(* Logix 5000 project; controller cal1632 1756-L62 rev 16.20; software revision 16.05; part 53 of 61 *)
(* tags used below, declared in another part *)
   turret_wa_pos_doff_request : BOOL;   // Turret Move to Winder A Doff Position Request
   turret_wa_pos_run_request : BOOL;   // Turret Move to Winder A Run Position
   turret_wb_pos_doff_request : BOOL;   // Turret Move to Winder B Doff Position Request
   turret_wb_pos_run_request : BOOL;   // Turret Move to Winder B Run Position
   any_jog_wa_permissive : BOOL;   // Winder A Any Jog Permissive
   any_jog_wb_permissive : BOOL;   // Winder B Any Jog Permissive
   di_mode_doff : BOOL;   // Doff Mode
   di_mode_run : BOOL;   // Run Mode
   FAULT : BOOL;
   HMI : BOOL;
   p00_wac_position_pct : REAL;   // Winder Accumulator Carriage Position Filtered [% of Stroke]
   p01_recipe_active : recipe;
   p01r09_pb_global_reset : BOOL;
   p01r13_line_running : BOOL;
   p01r13_line_slow_ramp : BOOL;
   p01r13_winder_tension_ok : BOOL;
   p02_real_from_hmi : hmi_real;
   p21r10_index_kd : REAL;
   p21r10_index_ki : REAL;
   p21r10_index_kp : REAL;
   p25_ao_selected_speed : REAL;
   p29_ai_wa_speed : REAL;
   p29_ai_wa_torque : REAL;
   p29_ai_wdr_lc : REAL;
   p29_di_wdr_a : BOOL;
   p29_di_wdr_index_fwd : BOOL;
   p29_dint_to_hmi : DINT[16];
   p29_param_acc_park_sp : REAL;   // Winder Accumulator Speed Trim Park Setpoint - Where the Carriage Sits [% of Stroke]
   p29_param_acc_trim_gain : REAL;   // Winder Accumulator Speed Trim Proportional Gain Fraction of Line Speed per % of Stroke
   p29_param_index_trim_fpm : REAL;
   p29_param_speed_trim_max : REAL;
   p29_param_speed_trim_min : REAL;   // Winder Accumulator Speed Trim Minimum - Fraction of Line Speed
   p29r01 : routine;
   p29r07 : routine;
   p29r07_timer_fault : TIMER[4];
   p29r07_timer_warning : TIMER[4];
   p29r08 : routine;
   p29r08_timer_fault : TIMER[4];
   p29r08_timer_warning : TIMER[4];
   p29r09 : routine;
   p29r09_mode_doff_auto : BOOL;   // Winder Mode Doff Position - AUTO Winder A/B doff PB indexes the turret to the preset doff position
   p29r09_mode_doff_manual : BOOL;   // Winder Mode Doff Position - MANUAL Operator jogs the turret to doff, doff PBs do nothing
   p29r09_tension_mode : BOOL;
   p29r09_timer_fault : TIMER[4];
   p29r09_timer_warning : TIMER[4];
   p29r09_torque_mode : BOOL;
   p29r09_winder_a_active : BOOL;
   p29r09_winder_b_active : BOOL;
   p29r10 : routine;
   p29r10_acc_pstn_error : REAL;   // Winder Winder A Accumulator Position Error position - park setpoint [% of Stroke]
   p29r10_accel_bias : REAL;
   p29r10_calc_speed_offset : REAL;
   p29r10_index_active : BOOL;
   p29r10_line_guard : REAL;   // Winder Accumulator Speed Trim Line speed, floored at 1.0 fpm for the divide
   p29r10_misc_index_factor : REAL;
   p29r10_param_psn_gain : REAL;
   p29r10_pid_out : REAL;
   p29r10_pid_psn : PID;
   p29r10_pid_psn_cv : REAL;
   p29r10_pid_psn_pv : REAL;
   p29r10_pid_torque : REAL;
   p29r10_pid_tq : PID;
   p29r10_pid_tq_cv : REAL;
   p29r10_psn_gain : REAL;
   p29r10_request_run : BOOL;
   p29r10_run_permissive : BOOL;
   p29r10_speed_offset : REAL;
   p29r10_tension_error : REAL;   // Winder Winder A Tension Error winder_tension_sp - Load Cell [lbf]
   p29r10_timer : TIMER[4];
   p29r10_timer_fault : TIMER[4];
   p29r10_timer_warning : TIMER[4];
   p29r10_trim_clamp : sys_Limit_Clamp;   // Winder Winder A Speed Trim Clamp
   p29r10_trim_hi : REAL;   // Winder Accumulator Speed Trim Upper limit in use this scan
   p29r10_trim_lo : REAL;   // Winder Accumulator Speed Trim Lower limit in use this scan
   p29r11 : routine;
   p29r15 : routine;
   p29r15_request_jog_fwd : BOOL;
   p29r15_state : DINT;
   p29r15_wdra_active : BOOL;
   p29r16 : routine;
   p29r16_request_jog_fwd : BOOL;
   p29r17 : routine;
   p29r20 : routine;
(* P29_Winder, continued *)

ROUTINE R07_Alarms   (* ladder *)
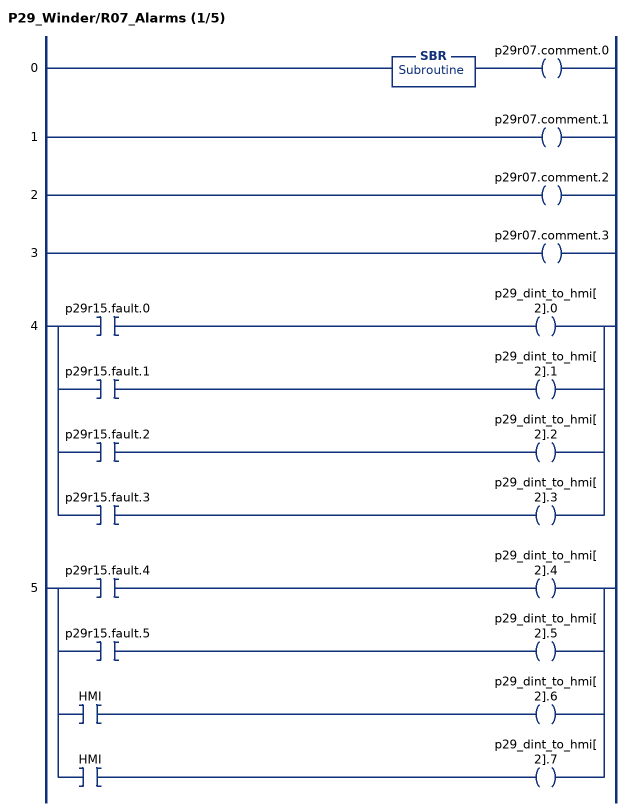
   0: SBR()OTE(p29r07.comment.0);
   1: OTE(p29r07.comment.1);
   2: OTE(p29r07.comment.2);
   3: OTE(p29r07.comment.3);
   4: [XIC(p29r15.fault.0) OTE(p29_dint_to_hmi[2].0) ,XIC(p29r15.fault.1) OTE(p29_dint_to_hmi[2].1) ,XIC(p29r15.fault.2) OTE(p29_dint_to_hmi[2].2) ,XIC(p29r15.fault.3) OTE(p29_dint_to_hmi[2].3) ];
   5: [XIC(p29r15.fault.4) OTE(p29_dint_to_hmi[2].4) ,XIC(p29r15.fault.5) OTE(p29_dint_to_hmi[2].5) ,XIC(HMI) OTE(p29_dint_to_hmi[2].6) ,XIC(HMI) OTE(p29_dint_to_hmi[2].7) ];
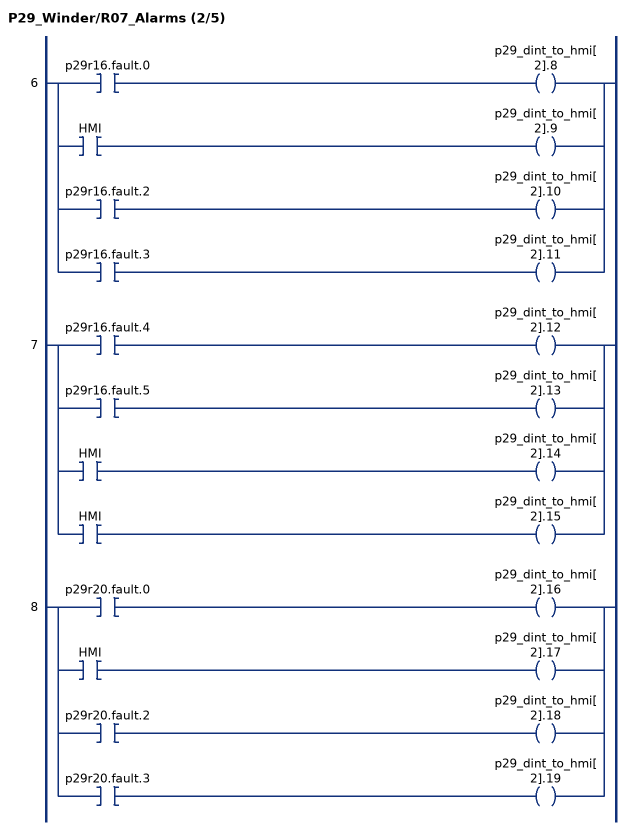
   6: [XIC(p29r16.fault.0) OTE(p29_dint_to_hmi[2].8) ,XIC(HMI) OTE(p29_dint_to_hmi[2].9) ,XIC(p29r16.fault.2) OTE(p29_dint_to_hmi[2].10) ,XIC(p29r16.fault.3) OTE(p29_dint_to_hmi[2].11) ];
   7: [XIC(p29r16.fault.4) OTE(p29_dint_to_hmi[2].12) ,XIC(p29r16.fault.5) OTE(p29_dint_to_hmi[2].13) ,XIC(HMI) OTE(p29_dint_to_hmi[2].14) ,XIC(HMI) OTE(p29_dint_to_hmi[2].15) ];
   8: [XIC(p29r20.fault.0) OTE(p29_dint_to_hmi[2].16) ,XIC(HMI) OTE(p29_dint_to_hmi[2].17) ,XIC(p29r20.fault.2) OTE(p29_dint_to_hmi[2].18) ,XIC(p29r20.fault.3) OTE(p29_dint_to_hmi[2].19) ];
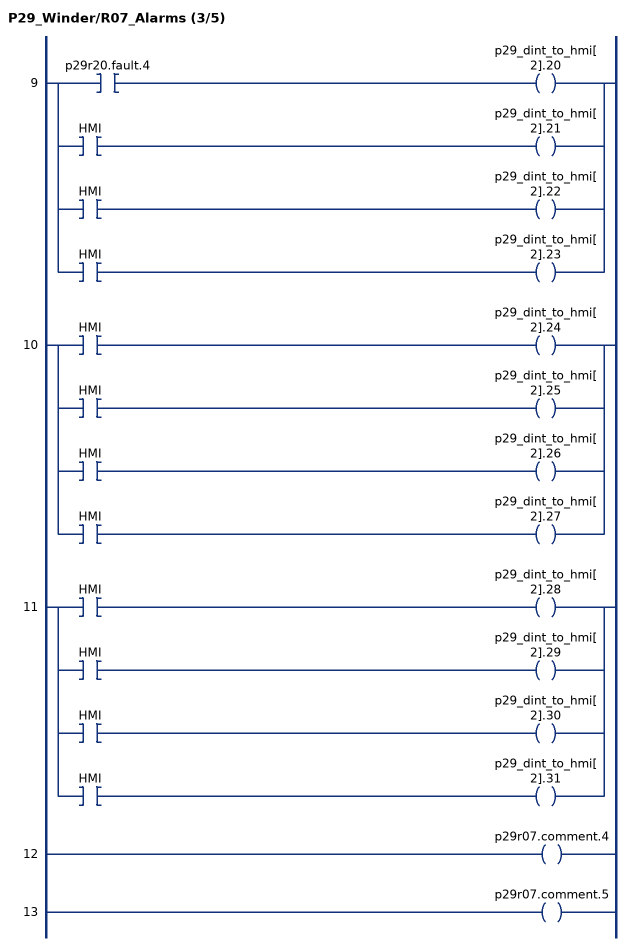
   9: [XIC(p29r20.fault.4) OTE(p29_dint_to_hmi[2].20) ,XIC(HMI) OTE(p29_dint_to_hmi[2].21) ,XIC(HMI) OTE(p29_dint_to_hmi[2].22) ,XIC(HMI) OTE(p29_dint_to_hmi[2].23) ];
   10: [XIC(HMI) OTE(p29_dint_to_hmi[2].24) ,XIC(HMI) OTE(p29_dint_to_hmi[2].25) ,XIC(HMI) OTE(p29_dint_to_hmi[2].26) ,XIC(HMI) OTE(p29_dint_to_hmi[2].27) ];
   11: [XIC(HMI) OTE(p29_dint_to_hmi[2].28) ,XIC(HMI) OTE(p29_dint_to_hmi[2].29) ,XIC(HMI) OTE(p29_dint_to_hmi[2].30) ,XIC(HMI) OTE(p29_dint_to_hmi[2].31) ];
   12: OTE(p29r07.comment.4);
   13: OTE(p29r07.comment.5);
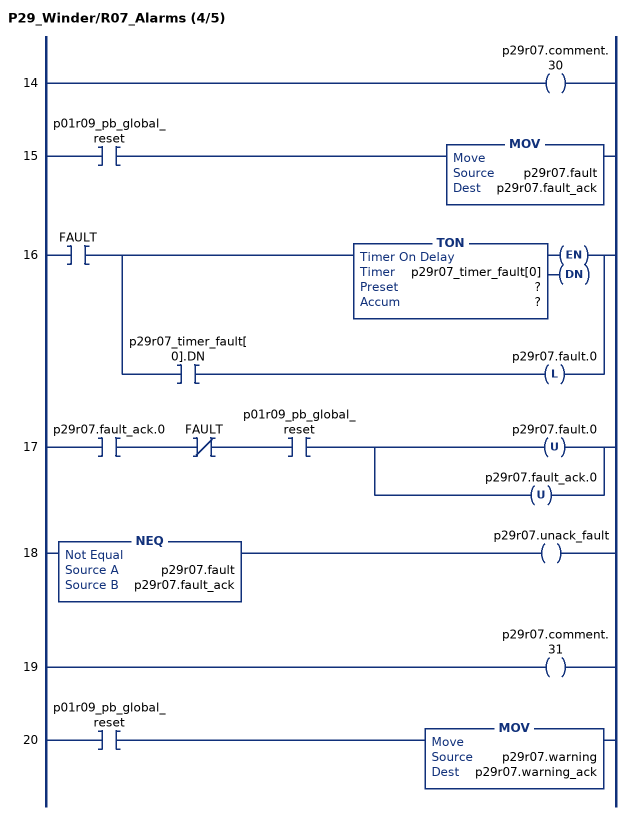
   14: OTE(p29r07.comment.30);
   15: XIC(p01r09_pb_global_reset)MOV(p29r07.fault,p29r07.fault_ack);
   16: XIC(FAULT)[TON(p29r07_timer_fault[0],?,?) ,XIC(p29r07_timer_fault[0].DN) OTL(p29r07.fault.0) ];
   17: XIC(p29r07.fault_ack.0)XIO(FAULT)XIC(p01r09_pb_global_reset)[OTU(p29r07.fault.0) ,OTU(p29r07.fault_ack.0) ];
   18: NEQ(p29r07.fault,p29r07.fault_ack)OTE(p29r07.unack_fault);
   19: OTE(p29r07.comment.31);
   20: XIC(p01r09_pb_global_reset)MOV(p29r07.warning,p29r07.warning_ack);
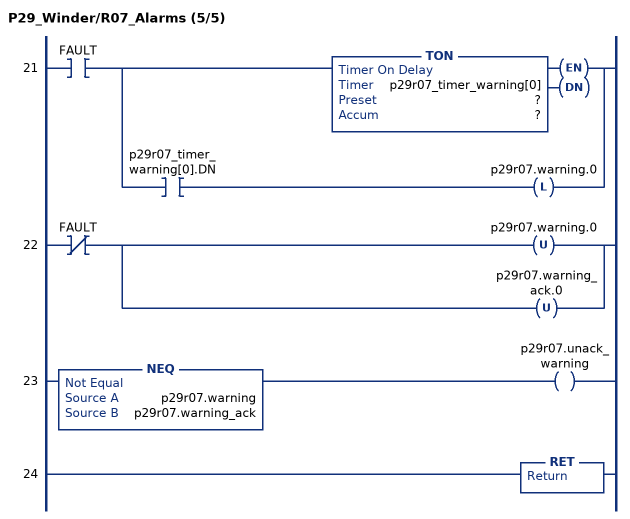
   21: XIC(FAULT)[TON(p29r07_timer_warning[0],?,?) ,XIC(p29r07_timer_warning[0].DN) OTL(p29r07.warning.0) ];
   22: XIO(FAULT)[OTU(p29r07.warning.0) ,OTU(p29r07.warning_ack.0) ];
   23: NEQ(p29r07.warning,p29r07.warning_ack)OTE(p29r07.unack_warning);
   24: RET();
END_ROUTINE

ROUTINE R08_Warnings   (* ladder *)
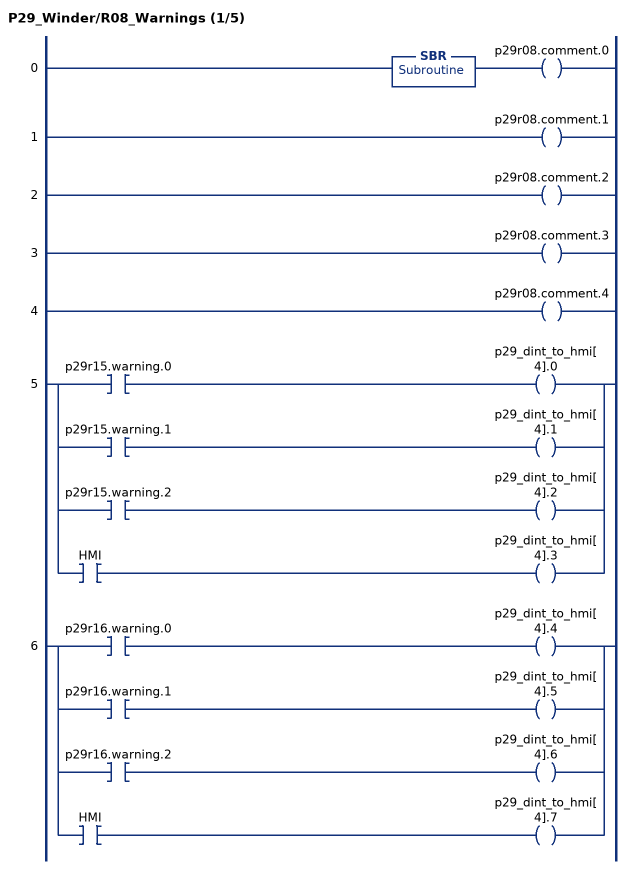
   0: SBR()OTE(p29r08.comment.0);
   1: OTE(p29r08.comment.1);
   2: OTE(p29r08.comment.2);
   3: OTE(p29r08.comment.3);
   4: OTE(p29r08.comment.4);
   5: [XIC(p29r15.warning.0) OTE(p29_dint_to_hmi[4].0) ,XIC(p29r15.warning.1) OTE(p29_dint_to_hmi[4].1) ,XIC(p29r15.warning.2) OTE(p29_dint_to_hmi[4].2) ,XIC(HMI) OTE(p29_dint_to_hmi[4].3) ];
   6: [XIC(p29r16.warning.0) OTE(p29_dint_to_hmi[4].4) ,XIC(p29r16.warning.1) OTE(p29_dint_to_hmi[4].5) ,XIC(p29r16.warning.2) OTE(p29_dint_to_hmi[4].6) ,XIC(HMI) OTE(p29_dint_to_hmi[4].7) ];
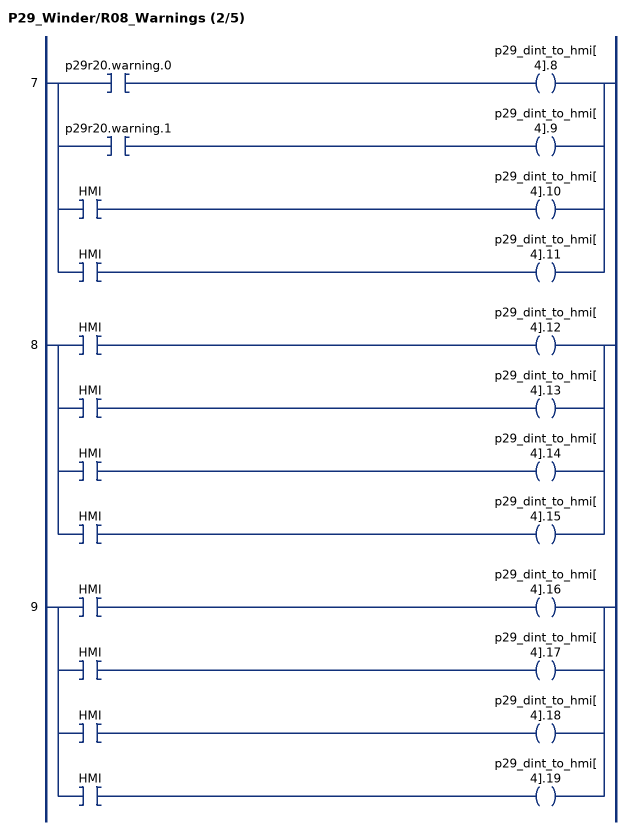
   7: [XIC(p29r20.warning.0) OTE(p29_dint_to_hmi[4].8) ,XIC(p29r20.warning.1) OTE(p29_dint_to_hmi[4].9) ,XIC(HMI) OTE(p29_dint_to_hmi[4].10) ,XIC(HMI) OTE(p29_dint_to_hmi[4].11) ];
   8: [XIC(HMI) OTE(p29_dint_to_hmi[4].12) ,XIC(HMI) OTE(p29_dint_to_hmi[4].13) ,XIC(HMI) OTE(p29_dint_to_hmi[4].14) ,XIC(HMI) OTE(p29_dint_to_hmi[4].15) ];
   9: [XIC(HMI) OTE(p29_dint_to_hmi[4].16) ,XIC(HMI) OTE(p29_dint_to_hmi[4].17) ,XIC(HMI) OTE(p29_dint_to_hmi[4].18) ,XIC(HMI) OTE(p29_dint_to_hmi[4].19) ];
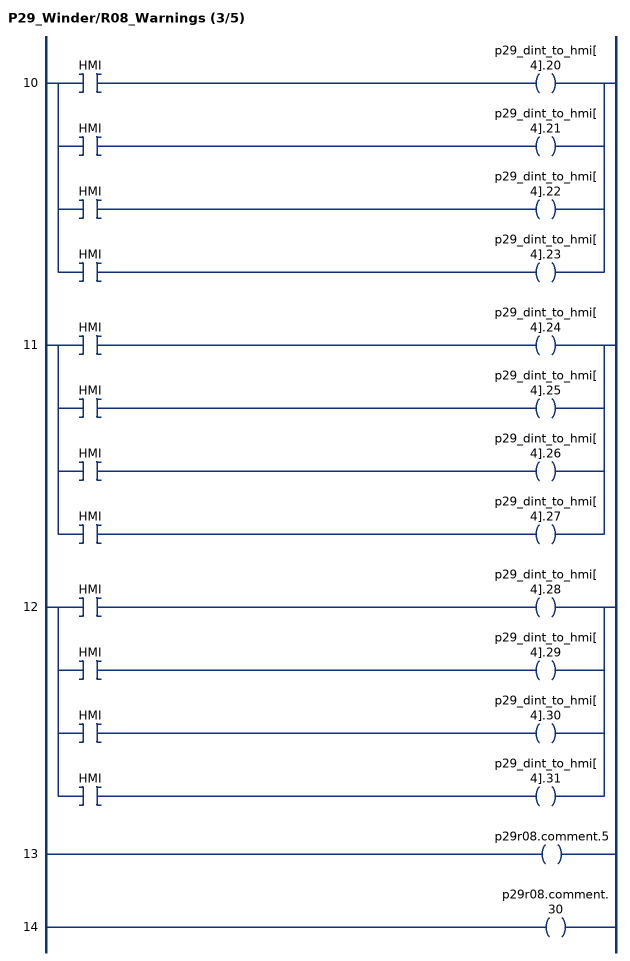
   10: [XIC(HMI) OTE(p29_dint_to_hmi[4].20) ,XIC(HMI) OTE(p29_dint_to_hmi[4].21) ,XIC(HMI) OTE(p29_dint_to_hmi[4].22) ,XIC(HMI) OTE(p29_dint_to_hmi[4].23) ];
   11: [XIC(HMI) OTE(p29_dint_to_hmi[4].24) ,XIC(HMI) OTE(p29_dint_to_hmi[4].25) ,XIC(HMI) OTE(p29_dint_to_hmi[4].26) ,XIC(HMI) OTE(p29_dint_to_hmi[4].27) ];
   12: [XIC(HMI) OTE(p29_dint_to_hmi[4].28) ,XIC(HMI) OTE(p29_dint_to_hmi[4].29) ,XIC(HMI) OTE(p29_dint_to_hmi[4].30) ,XIC(HMI) OTE(p29_dint_to_hmi[4].31) ];
   13: OTE(p29r08.comment.5);
   14: OTE(p29r08.comment.30);
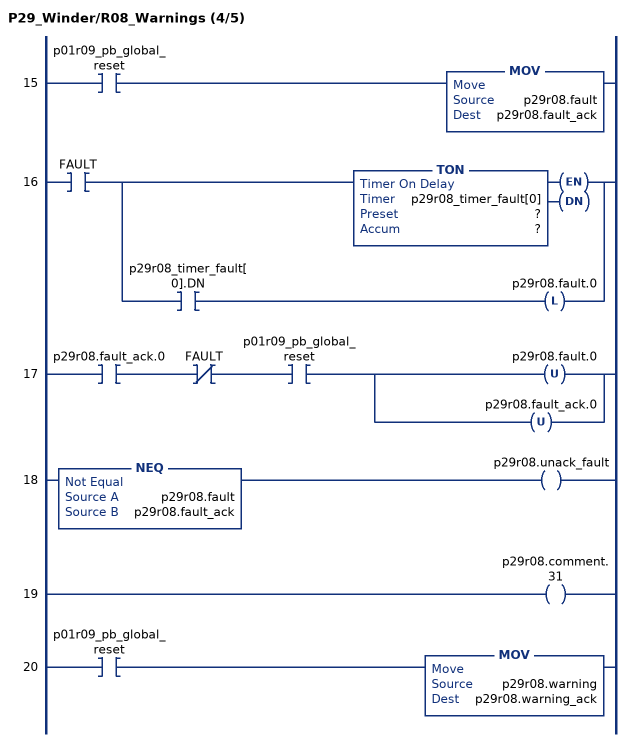
   15: XIC(p01r09_pb_global_reset)MOV(p29r08.fault,p29r08.fault_ack);
   16: XIC(FAULT)[TON(p29r08_timer_fault[0],?,?) ,XIC(p29r08_timer_fault[0].DN) OTL(p29r08.fault.0) ];
   17: XIC(p29r08.fault_ack.0)XIO(FAULT)XIC(p01r09_pb_global_reset)[OTU(p29r08.fault.0) ,OTU(p29r08.fault_ack.0) ];
   18: NEQ(p29r08.fault,p29r08.fault_ack)OTE(p29r08.unack_fault);
   19: OTE(p29r08.comment.31);
   20: XIC(p01r09_pb_global_reset)MOV(p29r08.warning,p29r08.warning_ack);
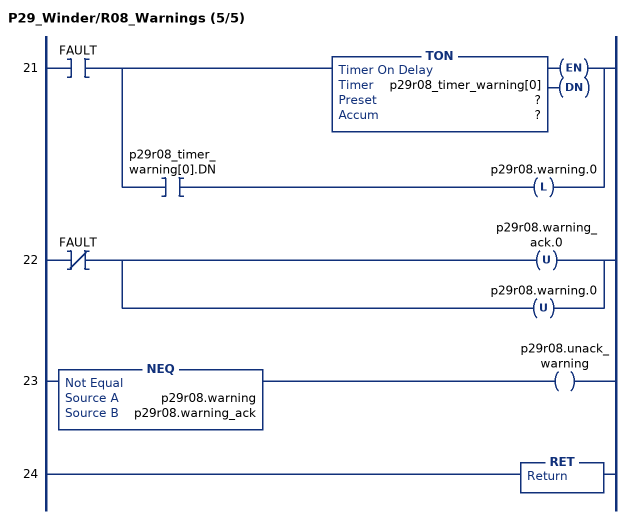
   21: XIC(FAULT)[TON(p29r08_timer_warning[0],?,?) ,XIC(p29r08_timer_warning[0].DN) OTL(p29r08.warning.0) ];
   22: XIO(FAULT)[OTU(p29r08.warning_ack.0) ,OTU(p29r08.warning.0) ];
   23: NEQ(p29r08.warning,p29r08.warning_ack)OTE(p29r08.unack_warning);
   24: RET();
END_ROUTINE

ROUTINE R09_Modes   (* ladder *)
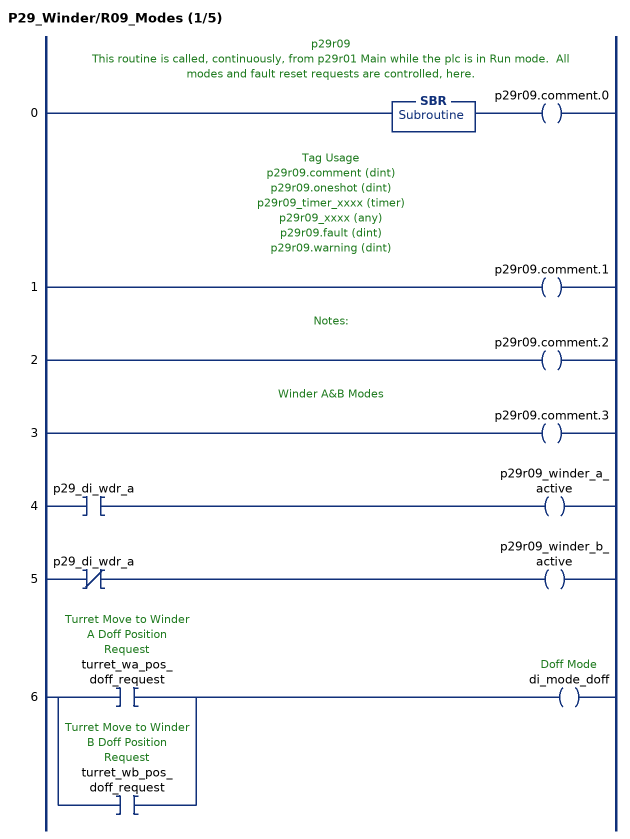
   // p29r09
   // This routine is called, continuously, from p29r01 Main while the plc is in Run mode.  All modes and fault reset requests are controlled, here.
   0: SBR()OTE(p29r09.comment.0);
   // Tag Usage
   // p29r09.comment (dint)
   // p29r09.oneshot (dint)
   // p29r09_timer_xxxx (timer)
   // p29r09_xxxx (any)
   // p29r09.fault (dint)
   // p29r09.warning (dint)
   1: OTE(p29r09.comment.1);
   // Notes:
   2: OTE(p29r09.comment.2);
   // Winder A&B Modes
   3: OTE(p29r09.comment.3);
   4: XIC(p29_di_wdr_a)OTE(p29r09_winder_a_active);
   5: XIO(p29_di_wdr_a)OTE(p29r09_winder_b_active);
   6: [XIC(turret_wa_pos_doff_request) ,XIC(turret_wb_pos_doff_request) ]OTE(di_mode_doff);
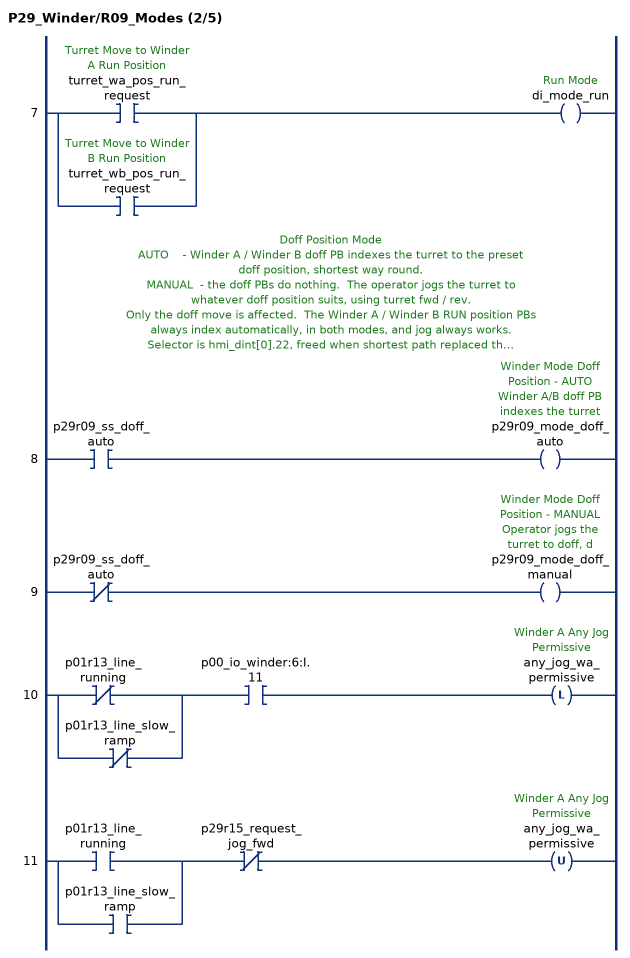
   7: [XIC(turret_wa_pos_run_request) ,XIC(turret_wb_pos_run_request) ]OTE(di_mode_run);
   // Doff Position Mode
   // AUTO    - Winder A / Winder B doff PB indexes the turret to the preset
   //           doff position, shortest way round.
   // MANUAL  - the doff PBs do nothing.  The operator jogs the turret to
   //           whatever doff position suits, using turret fwd / rev.
   // Only the doff move is affected.  The Winder A / Winder B RUN position PBs
   // always index automatically, in both modes, and jog always works.
   // Selector is hmi_dint[0].22, freed when shortest path replaced the
   // mode_under direction override.
   // Rev 20260825 a29
   8: XIC(p29r09_ss_doff_auto)OTE(p29r09_mode_doff_auto);
   9: XIO(p29r09_ss_doff_auto)OTE(p29r09_mode_doff_manual);
   10: [XIO(p01r13_line_running) ,XIO(p01r13_line_slow_ramp) ]XIC(p00_io_winder:6:I.11)OTL(any_jog_wa_permissive);
   11: [XIC(p01r13_line_running) ,XIC(p01r13_line_slow_ramp) ]XIO(p29r15_request_jog_fwd)OTU(any_jog_wa_permissive);
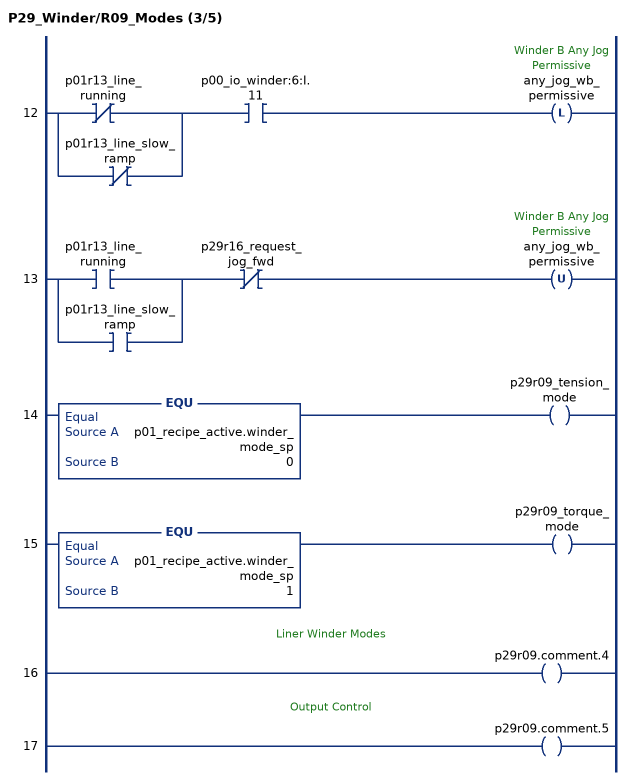
   12: [XIO(p01r13_line_running) ,XIO(p01r13_line_slow_ramp) ]XIC(p00_io_winder:6:I.11)OTL(any_jog_wb_permissive);
   13: [XIC(p01r13_line_running) ,XIC(p01r13_line_slow_ramp) ]XIO(p29r16_request_jog_fwd)OTU(any_jog_wb_permissive);
   14: EQU(p01_recipe_active.winder_mode_sp,0)OTE(p29r09_tension_mode);
   15: EQU(p01_recipe_active.winder_mode_sp,1)OTE(p29r09_torque_mode);
   // Liner Winder Modes
   16: OTE(p29r09.comment.4);
   // Output Control
   17: OTE(p29r09.comment.5);
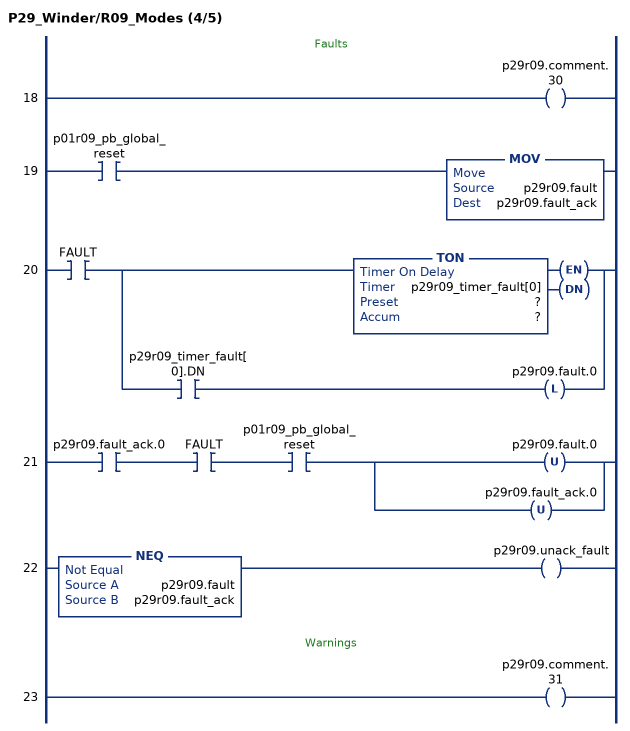
   // Faults
   18: OTE(p29r09.comment.30);
   19: XIC(p01r09_pb_global_reset)MOV(p29r09.fault,p29r09.fault_ack);
   20: XIC(FAULT)[TON(p29r09_timer_fault[0],?,?) ,XIC(p29r09_timer_fault[0].DN) OTL(p29r09.fault.0) ];
   21: XIC(p29r09.fault_ack.0)XIC(FAULT)XIC(p01r09_pb_global_reset)[OTU(p29r09.fault.0) ,OTU(p29r09.fault_ack.0) ];
   22: NEQ(p29r09.fault,p29r09.fault_ack)OTE(p29r09.unack_fault);
   // Warnings
   23: OTE(p29r09.comment.31);
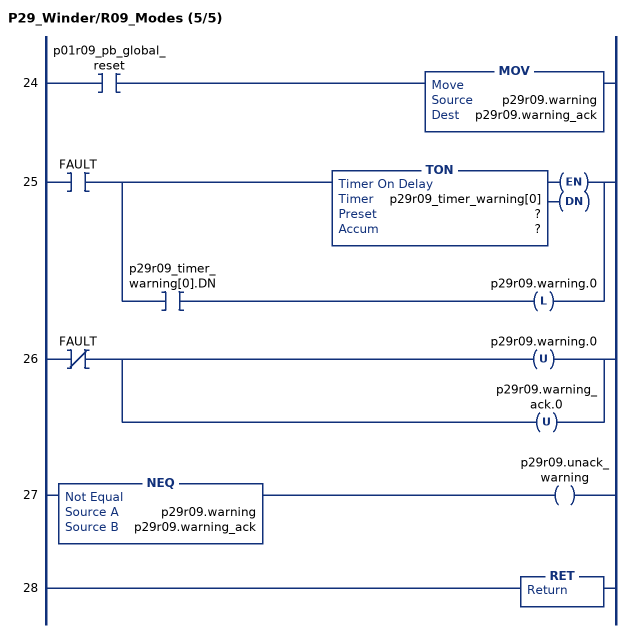
   24: XIC(p01r09_pb_global_reset)MOV(p29r09.warning,p29r09.warning_ack);
   25: XIC(FAULT)[TON(p29r09_timer_warning[0],?,?) ,XIC(p29r09_timer_warning[0].DN) OTL(p29r09.warning.0) ];
   26: XIO(FAULT)[OTU(p29r09.warning.0) ,OTU(p29r09.warning_ack.0) ];
   27: NEQ(p29r09.warning,p29r09.warning_ack)OTE(p29r09.unack_warning);
   28: RET();
END_ROUTINE

ROUTINE R10_Winder_A_Speed_Control   (* ladder *)
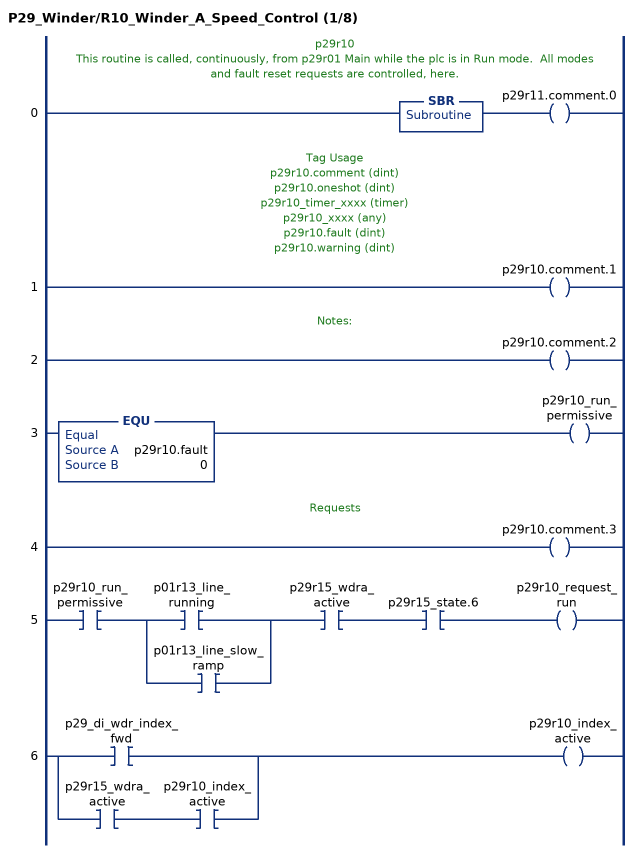
   // p29r10
   // This routine is called, continuously, from p29r01 Main while the plc is in Run mode.  All modes and fault reset requests are controlled, here.
   0: SBR()OTE(p29r11.comment.0);
   // Tag Usage
   // p29r10.comment (dint)
   // p29r10.oneshot (dint)
   // p29r10_timer_xxxx (timer)
   // p29r10_xxxx (any)
   // p29r10.fault (dint)
   // p29r10.warning (dint)
   1: OTE(p29r10.comment.1);
   // Notes:
   2: OTE(p29r10.comment.2);
   3: EQU(p29r10.fault,0)OTE(p29r10_run_permissive);
   // Requests
   4: OTE(p29r10.comment.3);
   5: XIC(p29r10_run_permissive)[XIC(p01r13_line_running) ,XIC(p01r13_line_slow_ramp) ]XIC(p29r15_wdra_active)XIC(p29r15_state.6)OTE(p29r10_request_run);
   6: [XIC(p29_di_wdr_index_fwd) ,XIC(p29r15_wdra_active) XIC(p29r10_index_active) ]OTE(p29r10_index_active);
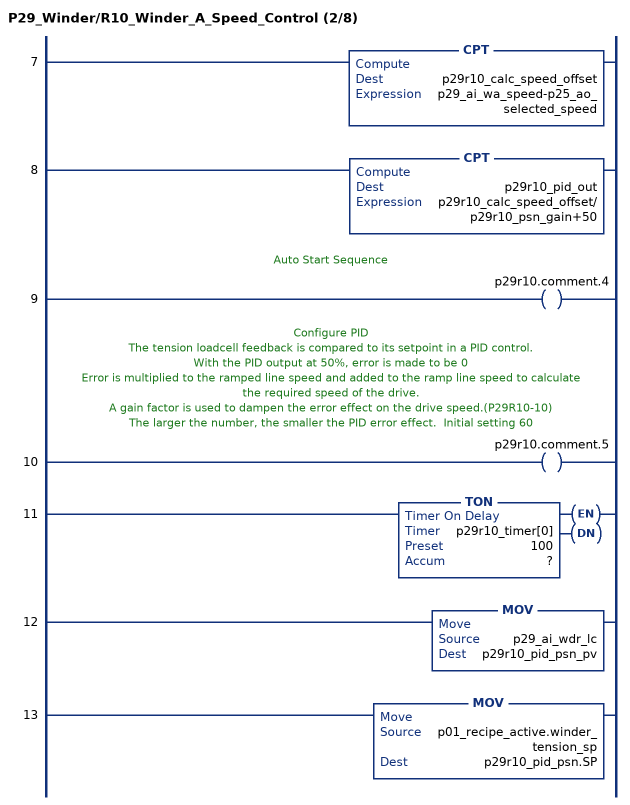
   7: CPT(p29r10_calc_speed_offset,p29_ai_wa_speed-p25_ao_selected_speed);
   8: CPT(p29r10_pid_out,p29r10_calc_speed_offset/p29r10_psn_gain+50);
   // Auto Start Sequence
   9: OTE(p29r10.comment.4);
   // Configure PID
   // The tension loadcell feedback is compared to its setpoint in a PID control.
   // With the PID output at 50%, error is made to be 0
   // Error is multiplied to the ramped line speed and added to the ramp line speed to calculate the required speed of the drive.
   // A gain factor is used to dampen the error effect on the drive speed.(P29R10-10)
   // The larger the number, the smaller the PID error effect.  Initial setting 60
   10: OTE(p29r10.comment.5);
   11: TON(p29r10_timer[0],?,?);
   12: MOV(p29_ai_wdr_lc,p29r10_pid_psn_pv);
   13: MOV(p01_recipe_active.winder_tension_sp,p29r10_pid_psn.SP);
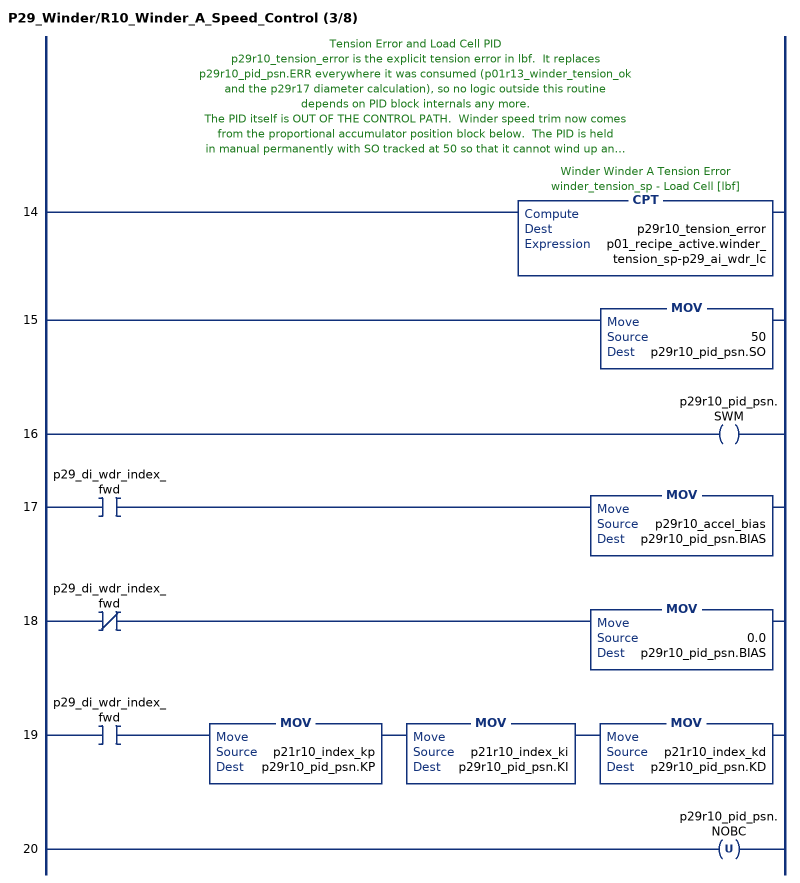
   // Tension Error and Load Cell PID
   // p29r10_tension_error is the explicit tension error in lbf.  It replaces
   // p29r10_pid_psn.ERR everywhere it was consumed (p01r13_winder_tension_ok
   // and the p29r17 diameter calculation), so no logic outside this routine
   // depends on PID block internals any more.
   // The PID itself is OUT OF THE CONTROL PATH.  Winder speed trim now comes
   // from the proportional accumulator position block below.  The PID is held
   // in manual permanently with SO tracked at 50 so that it cannot wind up and
   // the HMI faceplate shows a sane output.  Block and tags are kept declared
   // for HMI back-compat - delete the PID instruction if the faceplate goes.
   // Rev 20260820
   14: CPT(p29r10_tension_error,p01_recipe_active.winder_tension_sp-p29_ai_wdr_lc);
   15: MOV(50,p29r10_pid_psn.SO);
   16: OTE(p29r10_pid_psn.SWM);
   17: XIC(p29_di_wdr_index_fwd)MOV(p29r10_accel_bias,p29r10_pid_psn.BIAS);
   18: XIO(p29_di_wdr_index_fwd)MOV(0.0,p29r10_pid_psn.BIAS);
   19: XIC(p29_di_wdr_index_fwd)MOV(p21r10_index_kp,p29r10_pid_psn.KP)MOV(p21r10_index_ki,p29r10_pid_psn.KI)MOV(p21r10_index_kd,p29r10_pid_psn.KD);
   20: OTU(p29r10_pid_psn.NOBC);
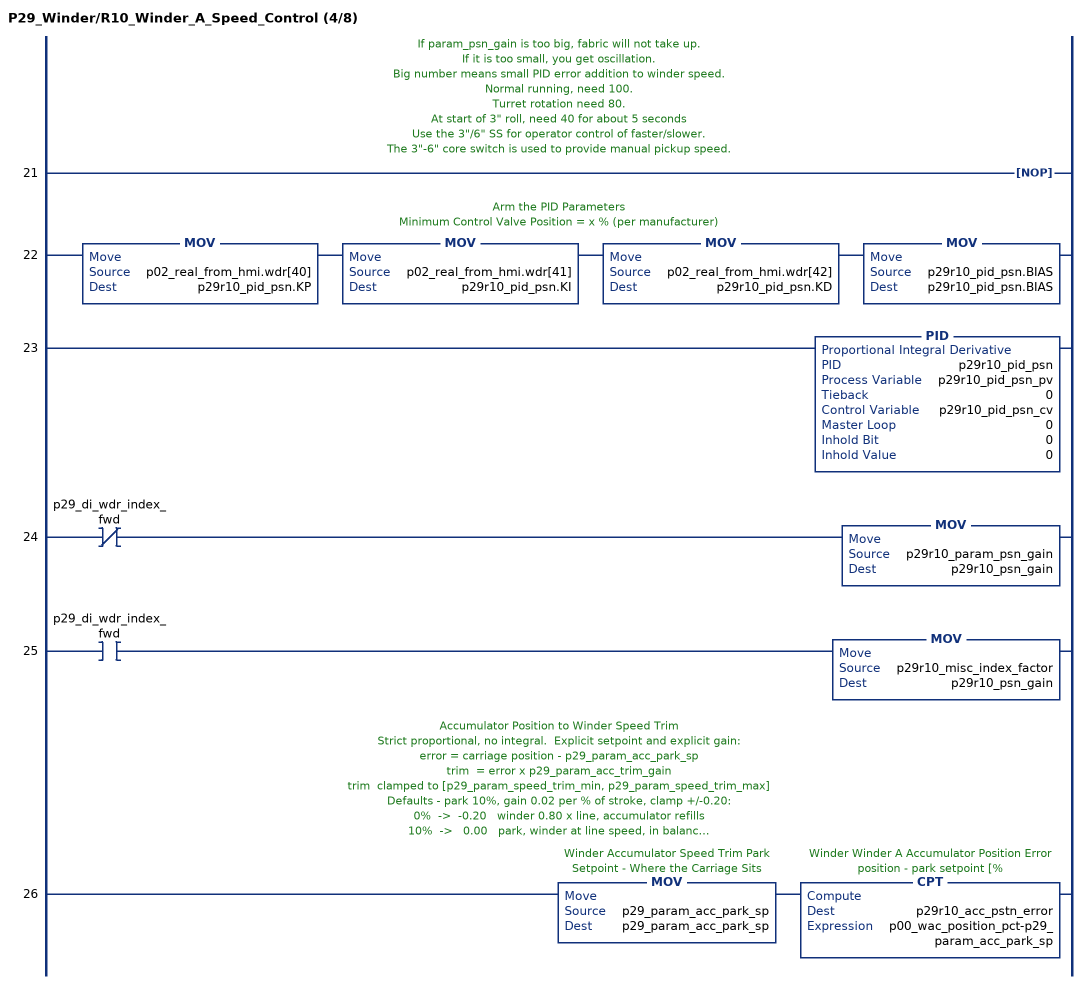
   // If param_psn_gain is too big, fabric will not take up.
   // If it is too small, you get oscillation.
   // Big number means small PID error addition to winder speed.
   // Normal running, need 100.
   // Turret rotation need 80.
   // At start of 3" roll, need 40 for about 5 seconds
   // Use the 3"/6" SS for operator control of faster/slower.
   // The 3"-6" core switch is used to provide manual pickup speed.
   21: NOP();
   // Arm the PID Parameters
   // Minimum Control Valve Position = x % (per manufacturer)
   22: MOV(p02_real_from_hmi.wdr[40],p29r10_pid_psn.KP)MOV(p02_real_from_hmi.wdr[41],p29r10_pid_psn.KI)MOV(p02_real_from_hmi.wdr[42],p29r10_pid_psn.KD)MOV(p29r10_pid_psn.BIAS,p29r10_pid_psn.BIAS);
   23: PID(p29r10_pid_psn,p29r10_pid_psn_pv,0,p29r10_pid_psn_cv,0,0,0);
   24: XIO(p29_di_wdr_index_fwd)MOV(p29r10_param_psn_gain,p29r10_psn_gain);
   25: XIC(p29_di_wdr_index_fwd)MOV(p29r10_misc_index_factor,p29r10_psn_gain);
   // Accumulator Position to Winder Speed Trim
   // Strict proportional, no integral.  Explicit setpoint and explicit gain:
   //    error = carriage position - p29_param_acc_park_sp
   //    trim  = error x p29_param_acc_trim_gain
   //    trim  clamped to [p29_param_speed_trim_min, p29_param_speed_trim_max]
   // Defaults - park 10%, gain 0.02 per % of stroke, clamp +/-0.20:
   //         0%  ->  -0.20   winder 0.80 x line, accumulator refills
   //        10%  ->   0.00   park, winder at line speed, in balance
   //        20%  ->  +0.20   winder 1.20 x line, drawing down
   //    above 20%  ->  +0.20  clamped - this IS the payout overspeed
   // Nothing commands the carriage to the park position.  Park is simply where
   // the trim crosses zero, and the loop settles there by negative feedback:
   // above park the winder outruns the line and the carriage falls, and the
   // trim shrinks as it approaches.  Steady state offset from park is
   // (persistent surface speed error) / gain - a 1% speed mismatch parks it
   // 0.5% of stroke off, and it clamps only at a 20% mismatch.
   // This replaces a SYS_SCP block that mapped 0-20% onto -0.20/+0.20.  That
   // worked, but the park position was implicit - it was the midpoint only
   // because the two trim limits were symmetric, so changing the negative
   // authority silently moved where the accumulator lived (trim_min -0.10 with
   // trim_max +0.20 would have parked it at 6.7%).  Setpoint, gain and
   // authority are now three independent parameters.
   // Why proportional only:  carriage position is the INTEGRAL of the speed
   // difference.  P on an integrating plant is a first order closed loop - it
   // cannot oscillate on its own and needs no integral term to remove offset.
   // It also holds no state, so there is no windup and no manual/auto handover.
   // If it ever hunts at high line speed, widen the band by REDUCING
   // p29_param_acc_trim_gain - do not reduce the trim clamp, that is the payout
   // authority and is now a separate number.
   // The load cell PID does not drive speed.  See the rungs above.
   // Rev 20260820 a02
   26: MOV(p29_param_acc_park_sp,p29_param_acc_park_sp)CPT(p29r10_acc_pstn_error,p00_wac_position_pct-p29_param_acc_park_sp);
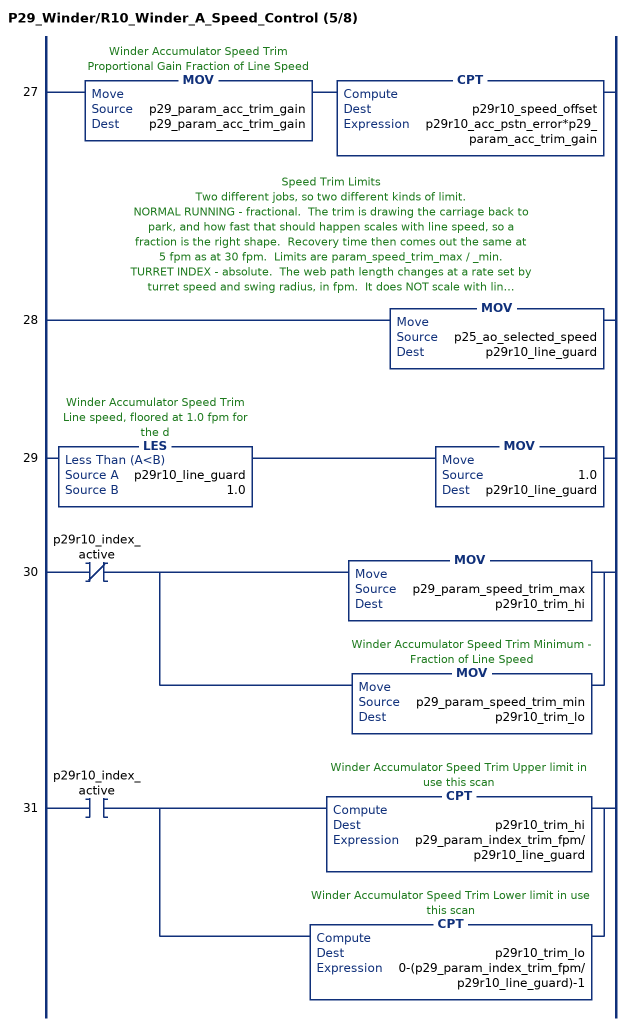
   27: MOV(p29_param_acc_trim_gain,p29_param_acc_trim_gain)CPT(p29r10_speed_offset,p29r10_acc_pstn_error*p29_param_acc_trim_gain);
   // Speed Trim Limits
   // Two different jobs, so two different kinds of limit.
   // NORMAL RUNNING - fractional.  The trim is drawing the carriage back to
   // park, and how fast that should happen scales with line speed, so a
   // fraction is the right shape.  Recovery time then comes out the same at
   // 5 fpm as at 30 fpm.  Limits are param_speed_trim_max / _min.
   // TURRET INDEX - absolute.  The web path length changes at a rate set by
   // turret speed and swing radius, in fpm.  It does NOT scale with line
   // speed.  A fraction is the wrong shape: 0.20 gives 6 fpm of authority at
   // 30 fpm line but only 1 fpm at 5 fpm line, where the disturbance is the
   // same size.  So during an index the limits become +/- the same absolute
   // fpm at any line speed:
   //   trim_hi =  index_trim_fpm / line     ->  winder = line + index_trim_fpm
   //   trim_lo = -index_trim_fpm / line - 1 ->  winder = -index_trim_fpm
   // trim_lo goes past -1 on purpose.  Below 1.0 the factor is negative and
   // the winder reverses, which it must be able to do: at the bottom of the
   // 5-30 fpm range the path lengthens faster than the line feeds.
   // line_guard floors the divisor at 1.0 fpm.  Line speed reaches 0 whenever
   // the line is stopped and this rung runs every scan.
   // Rev 20260825 a26
   28: MOV(p25_ao_selected_speed,p29r10_line_guard);
   29: LES(p29r10_line_guard,1.0)MOV(1.0,p29r10_line_guard);
   30: XIO(p29r10_index_active)[MOV(p29_param_speed_trim_max,p29r10_trim_hi) ,MOV(p29_param_speed_trim_min,p29r10_trim_lo) ];
   31: XIC(p29r10_index_active)[CPT(p29r10_trim_hi,p29_param_index_trim_fpm/p29r10_line_guard) ,CPT(p29r10_trim_lo,0-(p29_param_index_trim_fpm/p29r10_line_guard)-1) ];
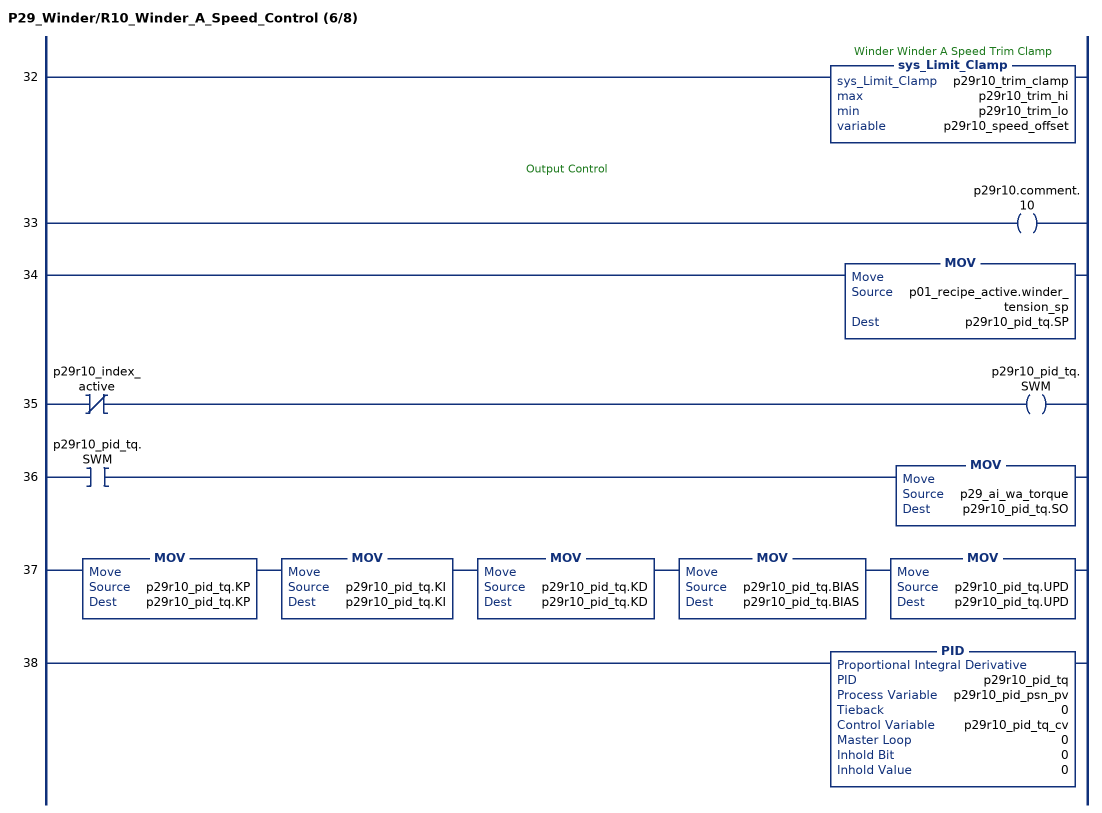
   32: sys_Limit_Clamp(p29r10_trim_clamp,p29r10_trim_hi,p29r10_trim_lo,p29r10_speed_offset);
   // Output Control
   33: OTE(p29r10.comment.10);
   34: MOV(p01_recipe_active.winder_tension_sp,p29r10_pid_tq.SP);
   35: XIO(p29r10_index_active)OTE(p29r10_pid_tq.SWM);
   36: XIC(p29r10_pid_tq.SWM)MOV(p29_ai_wa_torque,p29r10_pid_tq.SO);
   37: MOV(p29r10_pid_tq.KP,p29r10_pid_tq.KP)MOV(p29r10_pid_tq.KI,p29r10_pid_tq.KI)MOV(p29r10_pid_tq.KD,p29r10_pid_tq.KD)MOV(p29r10_pid_tq.BIAS,p29r10_pid_tq.BIAS)MOV(p29r10_pid_tq.UPD,p29r10_pid_tq.UPD);
   38: PID(p29r10_pid_tq,p29r10_pid_psn_pv,0,p29r10_pid_tq_cv,0,0,0);
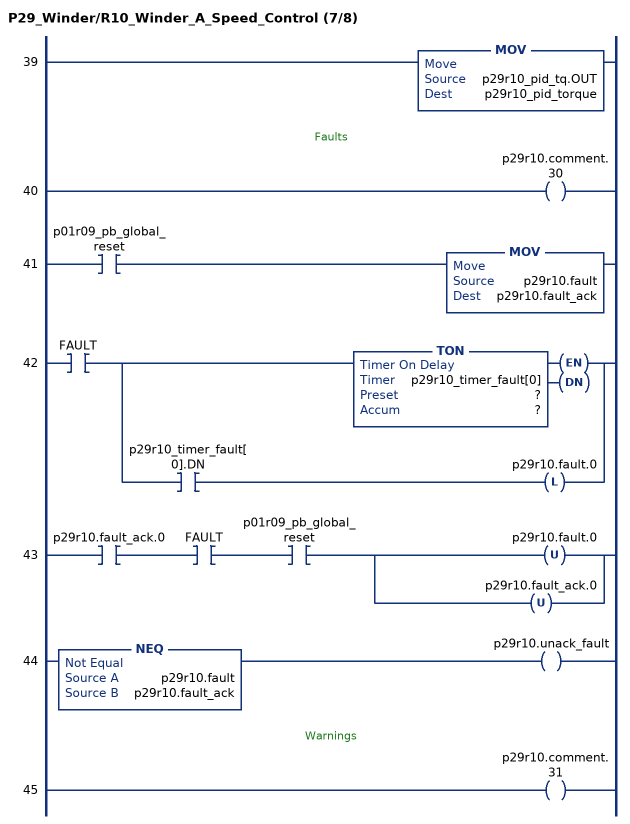
   39: MOV(p29r10_pid_tq.OUT,p29r10_pid_torque);
   // Faults
   40: OTE(p29r10.comment.30);
   41: XIC(p01r09_pb_global_reset)MOV(p29r10.fault,p29r10.fault_ack);
   42: XIC(FAULT)[TON(p29r10_timer_fault[0],?,?) ,XIC(p29r10_timer_fault[0].DN) OTL(p29r10.fault.0) ];
   43: XIC(p29r10.fault_ack.0)XIC(FAULT)XIC(p01r09_pb_global_reset)[OTU(p29r10.fault.0) ,OTU(p29r10.fault_ack.0) ];
   44: NEQ(p29r10.fault,p29r10.fault_ack)OTE(p29r10.unack_fault);
   // Warnings
   45: OTE(p29r10.comment.31);
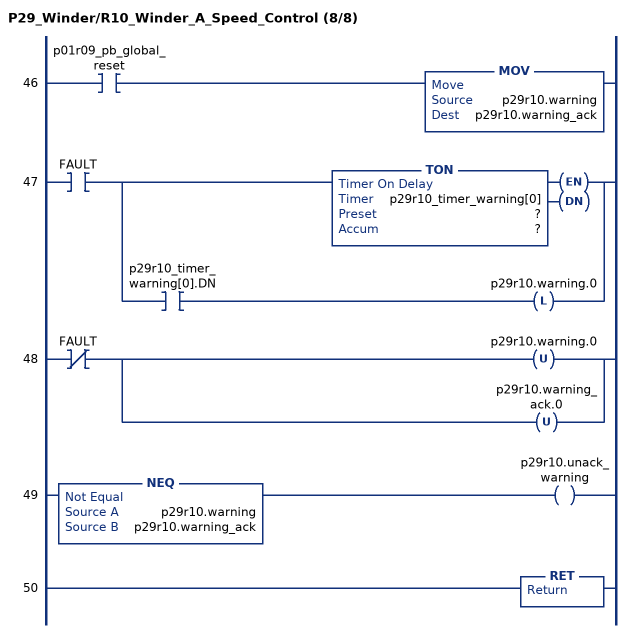
   46: XIC(p01r09_pb_global_reset)MOV(p29r10.warning,p29r10.warning_ack);
   47: XIC(FAULT)[TON(p29r10_timer_warning[0],?,?) ,XIC(p29r10_timer_warning[0].DN) OTL(p29r10.warning.0) ];
   48: XIO(FAULT)[OTU(p29r10.warning.0) ,OTU(p29r10.warning_ack.0) ];
   49: NEQ(p29r10.warning,p29r10.warning_ack)OTE(p29r10.unack_warning);
   50: RET();
END_ROUTINE
